{attribute 'GeneratedUsingTerminal: EL1252-0000-0018'}
{attribute addProperty BoxType "EL1252-0000-0018"}
{attribute addProperty Id "EtcSlaveTerminalBaseChannel_1AT %I*Channel_830843C11Channel_2AT %I*Channel_830843C11ReservedEMPTY_STRUCTURE0LatchAT %I*Latch_39BD7C7C34WcStateAT %I*WcState_9091E0EB2InfoDataAT %I*InfoData_A7436BC610"}
{attribute addProperty CRC "1730043865"}
{attribute addProperty Size "48"}
TYPE EL1252_671E5FD9 EXTENDS EtcSlaveTerminalBase :
STRUCT
	{attribute addProperty Name "Channel_1"}
	Channel_1 : Channel_830843C1;
	{attribute addProperty Name "Channel_2"}
	Channel_2 : Channel_830843C1;
	{attribute addProperty Name "Reserved"}
	Reserved : EMPTY_STRUCTURE;
	{attribute addProperty Name "Latch"}
	Latch : Latch_39BD7C7C;
	{attribute addProperty Name "WcState"}
	WcState : WcState_9091E0EB;
	{attribute addProperty Name "InfoData"}
	InfoData : InfoData_A7436BC6;
END_STRUCT
END_TYPE

(* stored: Version 1.2.0.0, ProductVersion 3.1.4024.9
   DUT EL1252_671E5FD9: Id {8a96e5a2-36b2-4b31-a009-6bc412680150} *)
